{attribute 'linkalways'} 
{attribute 'no_explicit_call' := 'This FB is a CLASS and must be accessed using methods or properties'}
{attribute 'enable_dynamic_creation'}
FUNCTION_BLOCK Node_F_VN_MinElementElementwise_TcVnPoint2_REAL EXTENDS VisionNode
VAR
    ipContainer : _ITcVnContainer;
    aMin : _TcVnPoint2_REAL;
    hrPrev : _HRESULT(S_OK);
    hresult : _HRESULT(S_OK);
END_VAR

METHOD PUBLIC  Clone : I_Node
VAR
	pNode : POINTER TO Node_F_VN_MinElementElementwise_TcVnPoint2_REAL;
END_VAR
pNode := __NEW(Node_F_VN_MinElementElementwise_TcVnPoint2_REAL);
Clone := pNode^;
END_METHOD

METHOD FB_init : BOOL
VAR_INPUT
	bInitRetains : BOOL; // if TRUE, the retain variables are initialized (warm start / cold start)
	bInCopyCode : BOOL;  // if TRUE, the instance afterwards gets moved into the copy code (online change)
END_VAR
AddInput('ipContainer', ipContainer);
AddInput('aMin', aMin);
AddInput('hrPrev', hrPrev);
AddOutput('ipContainer', ipContainer);
AddOutput('hresult',hresult);
END_METHOD

METHOD PROTECTED OnExecute : HRESULT
hresult.Value := F_VN_MinElementElementwise_TcVnPoint2_REAL(
    ipContainer := ipContainer.Value,
    aMin := aMin.Value,
    hrPrev:= hrPrev.Value);
END_METHOD

METHOD PUBLIC PreExecutionCheck
VAR_INPUT
	Check : I_PreExecutionChecks;
END_VAR
Check.IsTrue(ipContainer.IsValid, 'ipContainer must be a valid container');
END_METHOD

END_FUNCTION_BLOCK

(* stored: Version 1.1.0.1, ProductVersion 3.1.4024.13
   POU Node_F_VN_MinElementElementwise_TcVnPoint2_REAL: Id {85086fd7-2ff5-4b91-b0d3-308d87bf3d1f}, SpecialFunc None
   Folder Constructor: Id {dfbc9980-097c-47a1-ae7c-72b624455a83}
   Method Clone: Id {e1103924-a816-48f6-b3fe-52a3b0bd1ad4}
   Method FB_init: Id {5ed4837d-e031-4887-a36c-53f4e9201a42}
   Method OnExecute: Id {65561b4e-1438-4f66-a68b-ef2863742621}
   Method PreExecutionCheck: Id {38d6d6b8-9ec3-4500-8685-8ae97478f9c2} *)
